Fanuc KAREL source: COPY_FILE.kl

PROGRAM T
%NOLOCKGROUP
VAR
 v0 : STRING[40]
 v1 : STRING[40]
 v2 : BOOLEAN
 v3 : BOOLEAN
 v4 : INTEGER
BEGIN
 COPY_FILE(v0, v1, v2, v3, v4)
END T
